PROGRAM MAIN
VAR
	FB_AdsReadEvents_0		: Tc2_Utilities.FB_AdsReadEvents;
	aEvents: ARRAY [1..80] OF Tc2_Utilities.ST_ReadEvent;
	
	Events:ARRAY[1..4]	OF	Tc2_System.FB_SimpleAdsLogEvent;
	temp: REAL;
	ADSLOGEVENT_0: ADSLOGEVENT;
	CfgEvent: TcEvent;
	EventData:ST_EventData;
	TcEventDataFormatString : STRING    := '%f%d';
END_VAR

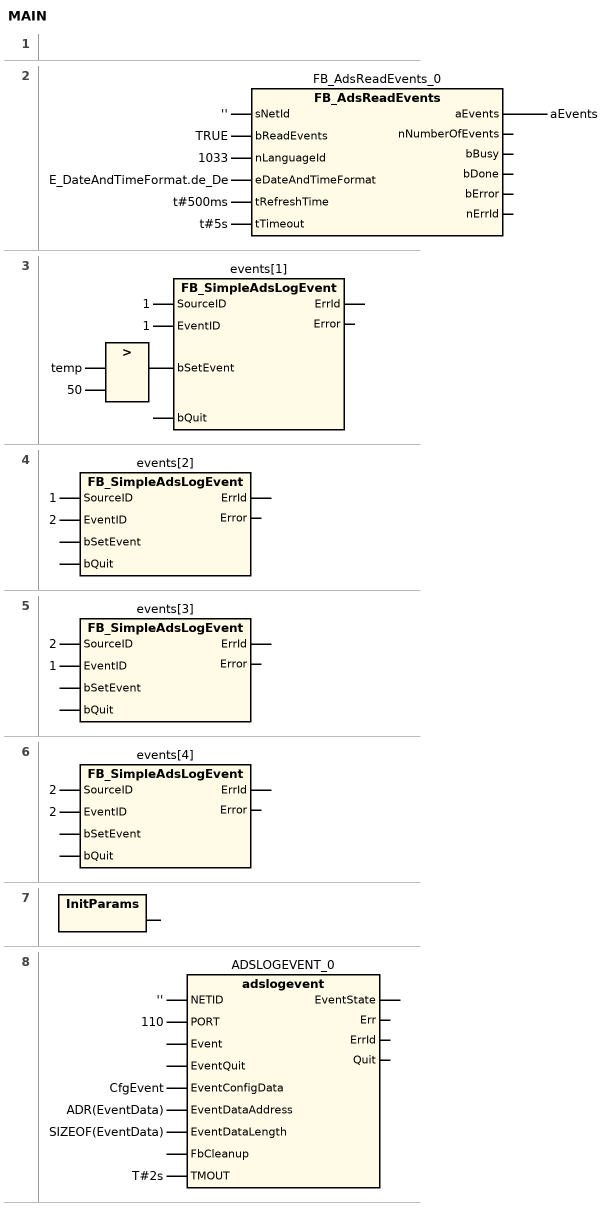
// NETWORK 1

// NETWORK 2
FB_AdsReadEvents_0(
    sNetId := '',
    bReadEvents := TRUE,
    nLanguageId := 1033,
    eDateAndTimeFormat := E_DateAndTimeFormat.de_De,
    tRefreshTime := t#500ms,
    tTimeout := t#5s); // FB_AdsReadEvents
aEvents := FB_AdsReadEvents_0.aEvents;

// NETWORK 3
events[1](SourceID := 1, EventID := 1, bSetEvent := temp > 50); // FB_SimpleAdsLogEvent

// NETWORK 4
events[2](SourceID := 1, EventID := 2); // FB_SimpleAdsLogEvent

// NETWORK 5
events[3](SourceID := 2, EventID := 1); // FB_SimpleAdsLogEvent

// NETWORK 6
events[4](SourceID := 2, EventID := 2); // FB_SimpleAdsLogEvent

// NETWORK 7
InitParams();

// NETWORK 8
ADSLOGEVENT_0(
    NETID := '',
    PORT := 110,
    EventConfigData := CfgEvent,
    EventDataAddress := ADR(EventData),
    EventDataLength := SIZEOF(EventData),
    TMOUT := T#2s); // adslogevent

ACTION InitParams:
//the folowing page explains settings in TcEvent
//https://infosys.beckhoff.com/content/1033/tcplclib_tc2_system/31081227.html?id=6547697951809802698



//CfgEvent.Class := TCEVENTCLASS_ALARM;
//CfgEvent.Prio := 2;
CfgEvent.Id := 1;
CfgEvent.SourceId := 3;
CfgEvent.bQuitRequired := TRUE;
CfgEvent.DataFormatStrAddress := ADR(TcEventDataFormatString);
CfgEvent.Flags := TCEVENTFLAG_LOG OR TCEVENTFLAG_SRCID OR TCEVENTFLAG_AUTOFMTALL;
CfgEvent.StreamType := TCEVENTSTREAM_SIMPLE;
//don't change this 
CfgEvent.ProgId :='TcEventFormatter.TcXMLFormatter' ;



//eventData.rVal     := 2.65;
//eventData.iVal    := 3;
END_ACTION

END_PROGRAM

(* stored: Version 1.1.0.1, ProductVersion 3.1.4024.11
   POU MAIN: Id {02be0bce-d303-4422-b4fe-406dee915a18}, SpecialFunc None
   Action InitParams: Id {03dd1058-903f-49e2-8ba1-185c6a9dd675} *)
